{attribute 'GeneratedUsingTerminal: ELM2642-0000-0016'}
{attribute addProperty BoxType "ELM2642-0000-0016"}
{attribute addProperty Id "Outputs_Channel_1AT %Q*Outputs_Channel_78994C084"}
{attribute addProperty CRC "117480092"}
{attribute addProperty Size "4"}
TYPE DO_Group_1_Outputs_07009A9C :
STRUCT
	{attribute addProperty Name "Outputs_Channel_1"}
	Outputs_Channel_1 AT %Q* : Outputs_Channel_78994C08;
END_STRUCT
END_TYPE

(* stored: Version 1.2.0.0, ProductVersion 3.1.4024.9
   DUT DO_Group_1_Outputs_07009A9C: Id {b22d1b8d-481a-4921-a575-2c71446417f1} *)
